TYPE TagsRedundancy :
STRUCT
	Settings: 	RedundancySettings; 	// Settings for the redundancy
	Status: 	RedundancyStatus; 		// Status for the redundancy
END_STRUCT
END_TYPE

(* stored: Version 1.1.0.1, ProductVersion 3.1.4024.6
   DUT TagsRedundancy: Id {e54e2645-0283-4cb7-8abf-1b06de56c2b7} *)
